PROGRAM prgEMS
VAR
	fbEMS1		: FB_EMS_V2;		//{#lynus.ag#()}
	fbEMS2		: FB_EMS_V2;		//{#lynus.ag#()}
END_VAR

//Fuse Line
fbEMS1.stNrOfEM_IN_ECS.diNrOfLine1 := prgUV.fbUV1_1.diNrOfEM_OUT;
fbEMS1.stNrOfEM_IN_ECS.diNrOfLine2 := prgUV.fbUV1_2.diNrOfEM_OUT;
fbEMS1.stNrOfEM_IN_ECS.diNrOfLine3 := prgUV.fbUV2_1.diNrOfEM_OUT;
fbEMS1.stNrOfEM_IN_ECS.diNrOfLine4 := prgUV.fbUV2_2.diNrOfEM_OUT;
fbEMS1.stNrOfEM_IN_ECS.diNrOfLine5 := prgUV.fbUV2_3.diNrOfEM_OUT;
fbEMS1.stNrOfEM_IN_ECS.diNrOfLine6 := prgUV.fbUV2_4.diNrOfEM_OUT;

fbEMS1(
	bEnable:= , 
	tDelayPwrCorrectionECS:= T#4S, 
	stNrOfEM_IN_ECS:= , 
	stSizeMainFuseCS:= , 
	stSetupEMS:= , 
	eOperationMode:= , 
	eSpeedModeBackendController:= E_SpeedModeBackendController_EMS.eSlow, 
	eSpeedModeLocalController:= E_SpeedModeLocalController_EMS.eSlow, 
	bActivateHP:= , 
	bControllingState:= , 
	rHeartbeat:= , 
	rErrorWarning:= , 
	rEnergyOptReady:= , 
	rNewBattPower:= , 
	eMessageEMS=> , 
	bStateEnable=> , 
	bStateAllowChrgFromGrid=> , 
	bMissingPowerData=> , 
	bSurplusAvailable=> , 
	bSEnableMainFuseFunc=> , 
	byProgress=> , 
	uiState_OUT=> , 
	diNrOfEMS_OUT=> , 
	arrMinPrioReached=> , 
	arrMaxPrioReached=> );

//Fuse Line
fbEMS2.stNrOfEM_IN_ECS.diNrOfLine1 := prgUV.fbUV3_1.diNrOfEM_OUT;
fbEMS2.stNrOfEM_IN_ECS.diNrOfLine2 := prgUV.fbUV3_2.diNrOfEM_OUT;
fbEMS2.stNrOfEM_IN_ECS.diNrOfLine3 := prgUV.fbUV3_3.diNrOfEM_OUT;
fbEMS2.stNrOfEM_IN_ECS.diNrOfLine4 := prgUV.fbUV3_4.diNrOfEM_OUT;
	
fbEMS2(
	bEnable:= , 
	tDelayPwrCorrectionECS:= T#4S, 
	stNrOfEM_IN_ECS:= , 
	stSizeMainFuseCS:= , 
	stSetupEMS:= , 
	eOperationMode:= , 
	eSpeedModeBackendController:= E_SpeedModeBackendController_EMS.eSlow, 
	eSpeedModeLocalController:= E_SpeedModeLocalController_EMS.eSlow, 
	bActivateHP:= , 
	bControllingState:= , 
	rHeartbeat:= , 
	rErrorWarning:= , 
	rEnergyOptReady:= , 
	rNewBattPower:= , 
	eMessageEMS=> , 
	bStateEnable=> , 
	bStateAllowChrgFromGrid=> , 
	bMissingPowerData=> , 
	bSurplusAvailable=> , 
	bSEnableMainFuseFunc=> , 
	byProgress=> , 
	uiState_OUT=> , 
	diNrOfEMS_OUT=> , 
	arrMinPrioReached=> , 
	arrMaxPrioReached=> );

END_PROGRAM

(* stored: Version 1.1.0.1, ProductVersion 3.1.4024.9
   POU prgEMS: Id {261512bd-8f5b-42a4-b98c-ad0de23e9cba}, SpecialFunc None *)
